PROGRAM POU_Manual_Auto
VAR
END_VAR

// NETWORK 1

END_PROGRAM

(* stored: Version 1.1.0.1, ProductVersion 3.1.4024.0
   POU POU_Manual_Auto: Id {8f5477e0-9e8e-40ab-9243-2cae32784338}, SpecialFunc None *)
